PROGRAM PRG_RestartService
// FB to Compress all files of the directory. 
VAR_INPUT
	IN_Directory			: T_MaxString; // directory of the file to compress
	ParamNetID				: STRING ; // Net ID of the PC with HH collector
	IN_ServiceName			: STRING  ;
	Start					: BOOL;
END_VAR
VAR
	StartProcess 			: NT_StartProcess;
	TrigStart				: R_TRIG;
END_VAR

TrigStart(CLK:=Start);
	StartProcess
	(
		NETID := ParamNetID,
		PATHSTR := concat(str1:= IN_Directory, str2 := 'IN_ServiceName'),
		DIRNAME := IN_Directory,
		COMNDLINE := '',
		Start := TrigStart.Q,
		TMOUT := T#3M
	);
	IF NOT StartProcess.BUSY THEN
		IF NOT StartProcess.ERR THEN
			StartProcess(Start := FALSE);
		ELSE
			StartProcess(Start := FALSE);
		END_IF
	END_IF

END_PROGRAM

(* stored: Version 1.1.0.1, ProductVersion 3.1.4024.6
   POU PRG_RestartService: Id {08ea3698-8b1f-4553-b646-92e832ba64ad}, SpecialFunc None *)
